PROGRAM TANKLEVEL
VAR CONSTANT
	L_S1:REAL :=  5.00 ;
	L_S2:REAL := 60.00 ;
	L_S3:REAL := 80.00 ;	
END_VAR

VAR
	Plant:FirstOrder;
	//fbNoise : FB_CTRL_NOISE_GENERATOR ;
	//fbNoiseParams : ST_CTRL_NOISE_GENERATOR_PARAMS ;
	//noise_level : LREAL ;
	fill_ValveA,fill_ValveB,Drain_ValveC: BOOL;
	fbdelayOFF:TOF;
// ---	
    fbFill, fbDrain : R_TRIG;
	fbFillOff, fbDrainOff :F_TRIG;
	currConstTime: REAL := 15;
	spLevel : REAL:=0;
    SensorNoise:fbSensorNoise;
END_VAR

// Generate sensor noise
//fbNoiseParams . tCtrlCycleTime := T#10MS ;
//fbNoiseParams . tTaskCycleTime := T#10MS ;
//fbNoiseParams . fAmplitude := 1.5 ;
//fbNoise ( fManSyncValue := 1 , eMode := 2 , stParams := fbNoiseParams ) ;
//noise_level := fbNoise.fOut ;
// Valves
Fill_ValveA := GVL_IO.ValveA ;
Fill_ValveB := GVL_IO.ValveB ;
Drain_ValveC := GVL_IO.ValveC ;

fbFill(clk := ( Fill_ValveA XOR Fill_ValveB ) AND NOT Drain_ValveC ) ;
fbFillOff(clk := Fill_ValveA XOR Fill_ValveB ) ;
fbDrain(clk := Drain_ValveC );
fbDrainOff(clk := Drain_ValveC );
fbdelayOFF(IN:=(GVL_IO.ValveA OR GVL_IO.ValveB OR GVL_IO.ValveC),PT:=T#1S);

IF fbFill.Q THEN
	spLevel:=150;
	currConstTime:=15;
END_IF
IF fbFillOff.Q THEN
	spLevel:=plant.fBOut;
	
END_IF
IF fbDrain.Q THEN
	currConstTime:=5;
    spLevel:=1;	
END_IF

IF fbDrainOff.Q THEN
	spLevel := GVL_IO.TankLevelSensor ;
END_IF

Plant(fBIn:= spLevel,Gain := 1,Tconstant := currConstTime);
SensorNoise(noise_enable:=TRUE,Ampl:=1.0);
//GVL_IO.TankLevelSensor:=plant.fBOut;
GVL_IO.TankLevelSensor:=LREAL_TO_REAL(plant.fBOut +SensorNoise.noise_level);
// IF (fbdelayOFF.Q) THEN
//	GVL_IO.TankLevelSensor:=LREAL_TO_REAL(plant.fBOut +SensorNoise.noise_level);
// END_IF
GVL_IO.Level_S1:=TRUE;
GVL_IO.Level_S2:=TRUE;
GVL_IO.Level_S3:=TRUE;

IF GVL_IO.TankLevelSensor > L_S1 THEN
	GVL_IO.Level_S1:=FALSE;
END_IF
IF GVL_IO.TankLevelSensor > L_S2 THEN
	GVL_IO.Level_S2:=FALSE;
END_IF
IF GVL_IO.TankLevelSensor > L_S3 THEN
	GVL_IO.Level_S3:=FALSE;
END_IF

 //

END_PROGRAM

(* stored: Version 1.1.0.1, ProductVersion 3.1.4024.2
   POU TANKLEVEL: Id {7d99a484-c811-47ca-b0f5-ff178effa6fa}, SpecialFunc None *)
